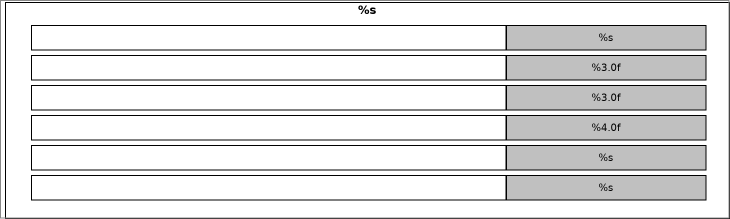
VISUALIZATION VISU_RECUPERATION_ETATS  // 730x219
VAR_IN_OUT
	COM: BLOCK_RS232_ONBOARD_V4;
END_VAR
    RoundedRectangle (5,2 725x217), "%s", text list: 'TextList_CryoPump', text index: 94
    Rectangle (506,55 200x25), "%3.0f", text variable: COM.STATE_Temperature[0]
    Rectangle (31,25 475x25), text list: 'TextList_CryoPump', text index: 4
    Rectangle (31,55 475x25), text list: 'TextList_CryoPump', text index: 5
    Rectangle (31,85 475x25), text list: 'TextList_CryoPump', text index: 6
    Rectangle (31,115 475x25), text list: 'TextList_CryoPump', text index: 53
    Rectangle (31,145 475x25), text list: 'TextList_CryoPump', text index: 39
    Rectangle (31,175 475x25), text list: 'TextList_CryoPump', text index: 40
    Rectangle (506,25 200x25), "%s", text variable: COM.PRM_PumpStartDelay, text list: 'TextList_CryoPump', text index: BOOL_TO_INT(COM.STATE_Pompe)+7
    Rectangle (506,85 200x25), "%3.0f", text variable: COM.STATE_Temperature[1]
    Rectangle (506,115 200x25), "%4.0f", text variable: COM.STATE_Pressure
    Rectangle (506,145 200x25), "%s", text list: 'TextList_CryoPump', text index: BOOL_TO_INT(COM.STATE_Rough_valve)+37
    Rectangle (506,175 200x25), "%s", text list: 'TextList_CryoPump', text index: BOOL_TO_INT(COM.STATE_Purge_valve)+37
END_VISUALIZATION

(* stored: Version 1.1.0.1, ProductVersion 3.1.4026.18
   Visu VISU_RECUPERATION_ETATS: Id {5805b743-4422-4908-9703-4be69a6b32f3} *)
